Omron Sysmac Studio project ExampleReadWriteVariables (Sysmac Studio 1.63.0.7, StandardProject)

# Controller Example: NX102-9000 version 1.64
Task PrimaryTask (priority 4, period or condition 4000): Main

VAR_GLOBAL
    WriteIntVal : DINT;  (* network input *)
    ReadIntVal : DINT;  (* network output *)
END_VAR

PROGRAM README
RETURN;
(*

# About This Project
This project is the server side program of PwshOpcUaClient.


# このプロジェクトについて
このプロジェクトは、PwshOpcUaClientのサーバ側プログラムです。


For the parts to which I have rights, I follow POU/Program/LICENSE.
You are free to use and modify it, but we are not responsible for any damage or loss related to it.

(c) 2025 KITA Munemitsu

*)
END_PROGRAM

PROGRAM Main
VAR
    iPrevWriteIntVal : DINT;
END_VAR
VAR_EXTERNAL
    WriteIntVal : DINT;
    ReadIntVal : DINT;
END_VAR
IF P_First_Run THEN
	iPrevWriteIntVal := WriteIntVal;
	ReadIntVal := 0;
END_IF;

IF WriteIntVal <> iPrevWriteIntVal THEN
	Inc(ReadIntVal);
	
	iPrevWriteIntVal := WriteIntVal;
END_IF;
END_PROGRAM

PROGRAM LICENSE
RETURN;
(*
The MIT License (MIT)

Copyright(c) 2025 KITA Munemitsu

Permission is hereby granted, free of charge, to any person obtaining a copy of this software and associated
documentation files (the “Software”), to deal in the Software without restriction, including without limitation
the rights to use, copy, modify, merge, publish, distribute, sublicense, and/or sell copies of the Software,
and to permit persons to whom the Software is furnished to do so, subject to the following conditions:

The above copyright notice and this permission notice shall be included in all copies or substantial portions of the Software.

THE SOFTWARE IS PROVIDED “AS IS”, WITHOUT WARRANTY OF ANY KIND, EXPRESS OR IMPLIED, INCLUDING BUT NOT
LIMITED TO THE WARRANTIES OF MERCHANTABILITY, FITNESS FOR A PARTICULAR PURPOSE AND NONINFRINGEMENT.
IN NO EVENT SHALL THE AUTHORS OR COPYRIGHT HOLDERS BE LIABLE FOR ANY CLAIM, DAMAGES OR OTHER LIABILITY,
WHETHER IN AN ACTION OF CONTRACT, TORT OR OTHERWISE, ARISING FROM, OUT OF OR IN CONNECTION WITH THE SOFTWARE
OR THE USE OR OTHER DEALINGS IN THE SOFTWARE.
*)
END_PROGRAM